FUNCTION F_ReadSimulatedTemperature : LREAL
VAR_STAT
	fbRand		: DRAND := (Seed:=TIME_TO_INT(TIME()));
END_VAR

fbRand();
F_ReadSimulatedTemperature := 20 + (fbRand.Num - 0.5) * 5;

END_FUNCTION

(* stored: Version 1.1.0.1, ProductVersion 3.1.4024.0
   POU F_ReadSimulatedTemperature: Id {4590c49e-4e3d-4064-95c4-9b0b8e156dfc}, SpecialFunc None *)
